# EPICS autosave request: support/ebrick/2-2-3/iocBoot/iocebrick/autosave/ebrickADC.req
$(P)$(H)$(F)$(D).SCAN
$(P)$(H)$(F)$(D).DESC
$(P)$(H)$(F)$(D).PREC
$(P)$(H)$(F)$(D).LOPR
$(P)$(H)$(F)$(D).HOPR
$(P)$(H)$(F)$(D).EGU
